/// configuration data that is used during boot to configure the Units equipment
TYPE QualityInspectionDataConfig :
STRUCT
  Simulated : BOOL;
END_STRUCT
END_TYPE

(* stored: Version 1.1.0.1
   DUT QualityInspectionDataConfig: Id {e5d3520b-7810-48b4-ac6f-a4592c8b7dc3} *)
